{attribute 'Tc2GvlVarNames'}
(* Generated automatically by TwinCAT - (read only) *)
VAR_CONFIG
	MAIN.Axis1.PlcToNc AT %QB0 : PLCTONC_AXIS_REF;
	MAIN.Axis1.NcToPlc AT %IB0 : NCTOPLC_AXIS_REF;
END_VAR

(* stored: Version 1.1.0.1, ProductVersion 3.1.4020.12
   GVL TwinCAT_Configuration: Id {67e0e72c-b864-4d13-8726-014b8f5cd7b7} *)
